PROGRAM VisionProgram
VAR
	fbCamera1 : FB_Camera;
END_VAR

fbCamera1();

END_PROGRAM

(* stored: Version 1.1.0.1, ProductVersion 3.1.4024.12
   POU VisionProgram: Id {4e1ae225-1f58-4af9-b633-a5d65bcb7583}, SpecialFunc None *)
